// TIA Portal project "winda" (V17)

(* hardware
DEVICE "S7-1500/ET200MP station_1"  S7-1500 station
   slot 0: "Rail_0"  Rack  6ES7 590-1***0-0AA0
   slot 1: "PLC_1"  CPU 1513-1 PN  6ES7 513-1AL02-0AB0  V2.9
      slot 3: "CPU display_1"  6ES7591-1AA00-0AA0
      slot 32768: "PROFINET interface_1"  X1
         slot 32769: "Port_1"  X1 P1
         slot 32770: "Port_2"  X1 P2
      slot 34817: "Virtual CP interface port_1"  Virtual CP interface port  Virtual CP interface port
*)

// ===== PLC "PLC_1"  CPU 1513-1 PN =====

VAR_GLOBAL   // PLC tag table "Default tag table"
   "wybrane" AT %MW50 : Int;
   "aktualne" AT %MW52 : Int;
   "jazda_dol" AT %Q0.0 : Bool;
   "jazda_gora" AT %Q0.1 : Bool;
   "Tag_5" AT %M50.0 : Bool;
   "Tag_6" AT %I0.0 : Bool;
   "Tag_7" AT %I0.1 : Bool;
   "Tag_8" AT %I0.2 : Bool;
   "Tag_9" AT %I0.3 : Bool;
   "Tag_10" AT %MW51 : Int;
   "T1Q" AT %M54.0 : Bool;
   "Tag_1" AT %M54.1 : Bool;
END_VAR

DATA_BLOCK "winda_LAD_DB"   // DB3
{ S7_Optimized_Access := 'TRUE' }
VERSION : 0.1
// stored: InstanceOfName winda_LAD
"winda_LAD"
BEGIN
END_DATA_BLOCK

DATA_BLOCK "winda_graph_DB1"   // DB4
{ S7_Optimized_Access := 'TRUE' }
VERSION : 0.1
// stored: InstanceOfName winda_graph
"winda_graph"
BEGIN
END_DATA_BLOCK

// folder: System blocks/Program resources

DATA_BLOCK "IEC_Timer_0_DB_1"   // DB1
{ S7_Optimized_Access := 'TRUE' }
AUTHOR : Simatic
FAMILY : IEC
NAME : IEC_TMR
VERSION : 1.0
// stored: InstanceOfName IEC_TIMER
"IEC_TIMER"
BEGIN
END_DATA_BLOCK

DATA_BLOCK "IEC_Timer_0_DB"   // DB2
{ S7_Optimized_Access := 'TRUE' }
AUTHOR : Simatic
FAMILY : IEC
NAME : IEC_TMR
VERSION : 1.0
// stored: InstanceOfName IEC_TIMER
"IEC_TIMER"
BEGIN
END_DATA_BLOCK

DATA_BLOCK "IEC_Timer_0_DB_2"   // DB5
{ S7_Optimized_Access := 'TRUE' }
AUTHOR : Simatic
FAMILY : IEC
NAME : IEC_TMR
VERSION : 1.0
// stored: InstanceOfName IEC_TIMER
"IEC_TIMER"
BEGIN
END_DATA_BLOCK

// folder: (top level)

FUNCTION_BLOCK "winda_graph"   // FB1, GRAPH_PLUS
{ S7_Optimized_Access := 'TRUE' }
VERSION : 0.1
   VAR_INPUT
      OFF_SQ : Bool := false;   // Turn sequence off
      INIT_SQ : Bool := false;   // Set sequence to initial state
      ACK_EF : Bool := false;   // Acknowledge all errors and faults
      S_PREV : Bool := false;   // Output previous step in parameter S_NO
      S_NEXT : Bool := false;   // Indicate next step in parameter S_NO
      SW_AUTO : Bool := false;   // Automatic mode
      SW_TAP : Bool := false;   // Semiautomatic/switch with transition
      SW_TOP : Bool := false;   // Semiautomatic/ignore transition
      SW_MAN : Bool := false;   // Manual mode
      S_SEL : Int := 0;   // Select step to be output to S_NO
      S_ON : Bool := false;   // Activate step indicated in S_NO
      S_OFF : Bool := false;   // Deactivate step indicated S_NO
      T_PUSH : Bool := false;   // Enable transition to switch in semi automatic mode
      aktualne_pietro : Int;
      wybrane_pietro : Int;
   END_VAR
   VAR_OUTPUT
      S_NO : Int := 0;   // Step number
      S_MORE : Bool := false;   // More steps are available and can be shown in S_NO
      S_ACTIVE : Bool := false;   // Step indicated in S_NO is active
      ERR_FLT : Bool := false;   // Interlock or supervision group error
      AUTO_ON : Bool := false;   // Automatic mode is active
      TAP_ON : Bool := false;   // Semiautomatic mode/step with transition enabled
      TOP_ON : Bool := false;   // Semiautomatic mode/ignore transition enabled
      MAN_ON : Bool := false;   // Manual mode is active
   END_VAR
   VAR_IN_OUT
      jedz_dol : Bool;
      jedz_gora : Bool;
   END_VAR
   VAR
      HMI_INFO : Array[0..8] of UInt;
      IF_PAR : G7_IfParPlus_V6;
      RT_DATA : G7_RTDataPlus_V6;   // Internal data area
      Trans1 : G7_TransitionPlus_V6;   // Transition structure
      Trans2 : G7_TransitionPlus_V6;   // Transition structure
      Trans3 : G7_TransitionPlus_V6;   // Transition structure
      Trans4 : G7_TransitionPlus_V6;   // Transition structure
      Trans6 : G7_TransitionPlus_V6;   // Transition structure
      Trans8 : G7_TransitionPlus_V6;   // Transition structure
      START : G7_StepPlus_V6;   // Step structure
      JAZDA_GORA : G7_StepPlus_V6;   // Step structure
      STOP_WINDY : G7_StepPlus_V6;   // Step structure
      JAZDA_DOL : G7_StepPlus_V6;   // Step structure
      STOP_WINDY2 : G7_StepPlus_V6;   // Step structure
      SINI : Array[0..1] of USInt;
      LSTT : Array[0..5] of USInt;
      ATAJ : Array[0..5] of USInt;
      ATAB : Array[0..5] of USInt;
      PSTT : Array[0..5] of USInt;
      NSTT : Array[0..5] of USInt;
      ASSJ : Array[0..4] of USInt;
      ASSB : Array[0..4] of USInt;
      PTTS : Array[0..4] of USInt;
      NTTS : Array[0..4] of USInt;
      SW_SQTS : Array[0..4] of USInt;
      SWITCH : Array[0..1] of USInt;
      TVX : Array[0..3] of USInt;
      TTX : Array[0..3] of USInt;
      TSX : Array[0..1] of USInt;
      S00X : Array[0..1] of USInt;
      SOFFX : Array[0..1] of USInt;
      SONX : Array[0..1] of USInt;
      SAX : Array[0..1] of USInt;
      SERRX : Array[0..5] of USInt;
      SMX : Array[0..5] of USInt;
      S0X : Array[0..5] of USInt;
      S1X : Array[0..5] of USInt;
      IL_ALARM_INST : Diag_Alarm;
      SUP_ALARM_INST : Diag_Alarm;
      STEP_TIME_ALARM_INST : Diag_Alarm;
      IEC_TIMER_INST : IEC_TIMER;
      TRANSACTION_FLAG : Bool := false;
   END_VAR
   // SINI[0] := 2;
   // LSTT[0] := 255;
   // LSTT[1] := 255;
   // LSTT[2] := 255;
   // LSTT[4] := 255;
   // ATAJ[1] := 1;
   // ATAJ[2] := 2;
   // ATAJ[3] := 3;
   // ATAJ[4] := 4;
   // ATAJ[5] := 5;
   // ATAB[0] := 1;
   // ATAB[2] := 2;
   // ATAB[3] := 3;
   // ATAB[4] := 4;
   // ATAB[5] := 5;
   // PSTT[2] := 1;
   // PSTT[3] := 2;
   // PSTT[4] := 3;
   // PSTT[5] := 4;
   // NSTT[0] := 3;
   // NSTT[1] := 1;
   // NSTT[2] := 2;
   // NSTT[4] := 4;
   // ASSJ[1] := 1;
   // ASSJ[2] := 2;
   // ASSJ[3] := 3;
   // ASSJ[4] := 4;
   // ASSB[1] := 1;
   // ASSB[2] := 2;
   // ASSB[3] := 3;
   // ASSB[4] := 4;
   // PTTS[0] := 255;
   // PTTS[1] := 1;
   // PTTS[2] := 2;
   // PTTS[4] := 4;
   // NTTS[1] := 2;
   // NTTS[2] := 3;
   // NTTS[3] := 4;
   // NTTS[4] := 5;
   // SW_SQTS[1] := 1;
   // SW_SQTS[2] := 1;
   // SW_SQTS[3] := 2;
   // SW_SQTS[4] := 2;
   // TVX[0] := 16#1;
   // TTX[0] := 16#1;
   // TSX[0] := 16#1;
   // S00X[0] := 16#1;
   // SOFFX[0] := 16#1;
   // SONX[0] := 16#1;
   // SAX[0] := 16#1;
   // SERRX[0] := 16#1;
   // SMX[0] := 16#1;
   // S0X[0] := 16#1;
   // S1X[0] := 16#1;
BEGIN
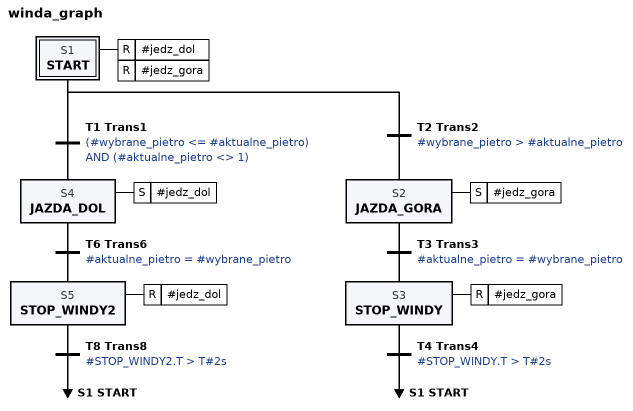
   // sequencer 1
   INITIAL_STEP START:   // S1, max time T#10S, warning time T#7S
              R    #jedz_dol
              R    #jedz_gora
   END_STEP
   TRANSITION Trans1 FROM START TO JAZDA_DOL   // T1
      := (#wybrane_pietro <= #aktualne_pietro) AND (#aktualne_pietro <> 1);
   END_TRANSITION
   TRANSITION Trans2 FROM START TO JAZDA_GORA   // T2
      := #wybrane_pietro > #aktualne_pietro;
   END_TRANSITION
   STEP JAZDA_GORA:   // S2, max time T#10S, warning time T#7S
              S    #jedz_gora
   END_STEP
   TRANSITION Trans3 FROM JAZDA_GORA TO STOP_WINDY   // T3
      := #aktualne_pietro = #wybrane_pietro;
   END_TRANSITION
   STEP STOP_WINDY:   // S3, max time T#10S, warning time T#7S
              R    #jedz_gora
   END_STEP
   TRANSITION Trans4 FROM STOP_WINDY TO START   // T4, jump
      := #STOP_WINDY.T > T#2s;
   END_TRANSITION
   STEP JAZDA_DOL:   // S4, max time T#10S, warning time T#7S
              S    #jedz_dol
   END_STEP
   TRANSITION Trans6 FROM JAZDA_DOL TO STOP_WINDY2   // T6
      := #aktualne_pietro = #wybrane_pietro;
   END_TRANSITION
   STEP STOP_WINDY2:   // S5, max time T#10S, warning time T#7S
              R    #jedz_dol
   END_STEP
   TRANSITION Trans8 FROM STOP_WINDY2 TO START   // T8, jump
      := #STOP_WINDY2.T > T#2s;
   END_TRANSITION
END_FUNCTION_BLOCK

FUNCTION_BLOCK "winda_LAD"   // FB2, LAD
{ S7_Optimized_Access := 'TRUE' }
VERSION : 0.1
   VAR_INPUT
      "1" : Bool;
      "2" : Bool;
      "3" : Bool;
      "4" : Bool;
   END_VAR
   VAR_IN_OUT
      aktualne_pietro : Int := 1;
      wybrane_pietro : Int := 1;
      jedz_dol : Bool;
      jedz_gora : Bool;
   END_VAR
   VAR
      START : Bool;
      JAZDA_DOL : Bool;
      JAZDA_GORA : Bool;
      "STOP WINDY" : Bool;
      kolejka : Array[0..3] of Bool;
      "1_static" : Bool;
      "2_static" : Bool;
      "3_static" : Bool;
      "4_static" : Bool;
   END_VAR
   VAR_TEMP
      v : Int;
   END_VAR
   VAR_TEMP   // added for the SCL form of the ladder/FBD networks
      _w1 : Bool;
      _w2 : Bool;
      _w3 : Bool;
      _w4 : Bool;
   END_VAR
BEGIN

REGION Network 1
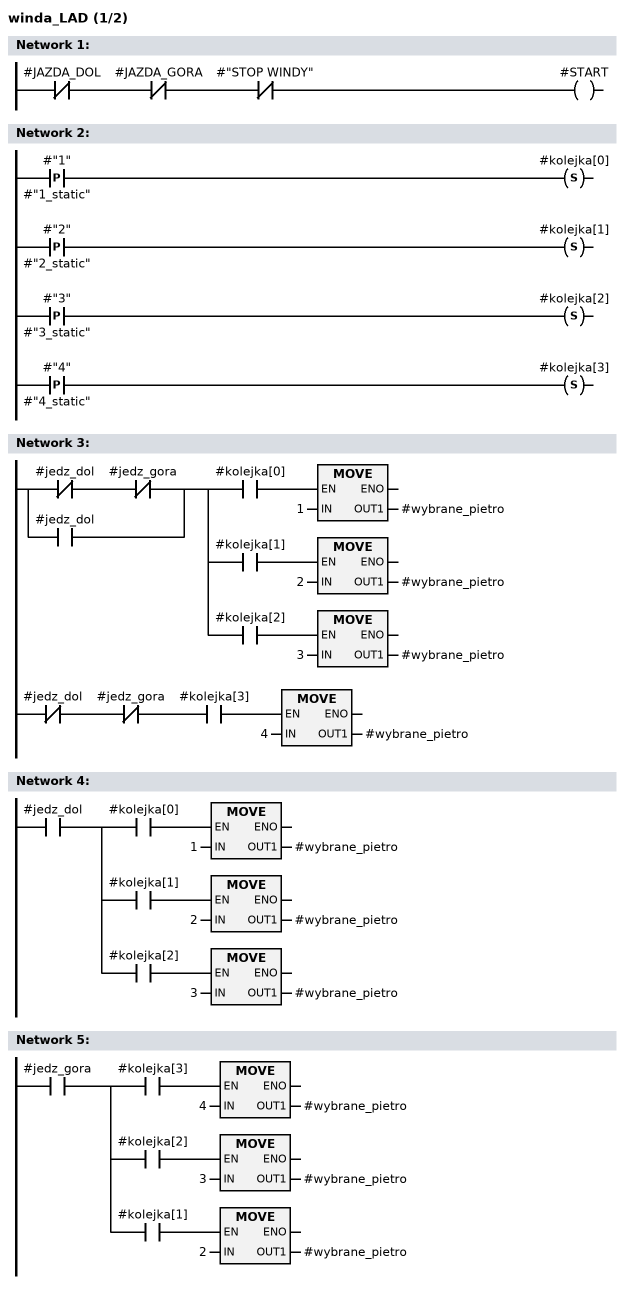
   RUNG wire#powerrail
      I_Contact( #JAZDA_DOL )
      I_Contact( #JAZDA_GORA )
      I_Contact( #"STOP WINDY" )
      Coil( #START )
   END_RUNG
   // the same network as SCL:
   #START := NOT #JAZDA_DOL AND NOT #JAZDA_GORA AND NOT #"STOP WINDY";
END_REGION

REGION Network 2
   RUNG wire#powerrail
      P_Contact(operand := #"1", bit := #"1_static")
      S_Coil( #kolejka[0] )
   END_RUNG
   RUNG wire#powerrail
      P_Contact(operand := #"2", bit := #"2_static")
      S_Coil( #kolejka[1] )
   END_RUNG
   RUNG wire#powerrail
      P_Contact(operand := #"3", bit := #"3_static")
      S_Coil( #kolejka[2] )
   END_RUNG
   RUNG wire#powerrail
      P_Contact(operand := #"4", bit := #"4_static")
      S_Coil( #kolejka[3] )
   END_RUNG
   // the same network as SCL:
   #_w1 := #"1" AND NOT #"1_static";   // rising edge of #"1"
   #"1_static" := #"1";
   IF #_w1 THEN #kolejka[0] := TRUE; END_IF;
   #_w2 := #"2" AND NOT #"2_static";   // rising edge of #"2"
   #"2_static" := #"2";
   IF #_w2 THEN #kolejka[1] := TRUE; END_IF;
   #_w3 := #"3" AND NOT #"3_static";   // rising edge of #"3"
   #"3_static" := #"3";
   IF #_w3 THEN #kolejka[2] := TRUE; END_IF;
   #_w4 := #"4" AND NOT #"4_static";   // rising edge of #"4"
   #"4_static" := #"4";
   IF #_w4 THEN #kolejka[3] := TRUE; END_IF;
END_REGION

REGION Network 3
   RUNG wire#powerrail
      I_Contact( #jedz_dol )
      I_Contact( #jedz_gora )
      wire#w1
      Contact( #kolejka[0] )
      Move(in := 1, out1 => #wybrane_pietro)
   END_RUNG
   RUNG wire#powerrail
      Contact( #jedz_dol )
   END_RUNG wire#w1
   RUNG wire#w1
      Contact( #kolejka[1] )
      Move(in := 2, out1 => #wybrane_pietro)
   END_RUNG
   RUNG wire#w1
      Contact( #kolejka[2] )
      Move(in := 3, out1 => #wybrane_pietro)
   END_RUNG
   RUNG wire#powerrail
      I_Contact( #jedz_dol )
      I_Contact( #jedz_gora )
      Contact( #kolejka[3] )
      Move(in := 4, out1 => #wybrane_pietro)
   END_RUNG
   // the same network as SCL:
   #_w1 := (NOT #jedz_dol AND NOT #jedz_gora) OR #jedz_dol;
   IF #_w1 AND #kolejka[0] THEN #wybrane_pietro := 1; END_IF;
   IF #_w1 AND #kolejka[1] THEN #wybrane_pietro := 2; END_IF;
   IF #_w1 AND #kolejka[2] THEN #wybrane_pietro := 3; END_IF;
   IF NOT #jedz_dol AND NOT #jedz_gora AND #kolejka[3] THEN #wybrane_pietro := 4; END_IF;
END_REGION

REGION Network 4
   RUNG wire#powerrail
      Contact( #jedz_dol )
      wire#w1
      Contact( #kolejka[0] )
      Move(in := 1, out1 => #wybrane_pietro)
   END_RUNG
   RUNG wire#w1
      Contact( #kolejka[1] )
      Move(in := 2, out1 => #wybrane_pietro)
   END_RUNG
   RUNG wire#w1
      Contact( #kolejka[2] )
      Move(in := 3, out1 => #wybrane_pietro)
   END_RUNG
   // the same network as SCL:
   IF #jedz_dol AND #kolejka[0] THEN #wybrane_pietro := 1; END_IF;
   IF #jedz_dol AND #kolejka[1] THEN #wybrane_pietro := 2; END_IF;
   IF #jedz_dol AND #kolejka[2] THEN #wybrane_pietro := 3; END_IF;
END_REGION

REGION Network 5
   RUNG wire#powerrail
      Contact( #jedz_gora )
      wire#w1
      Contact( #kolejka[3] )
      Move(in := 4, out1 => #wybrane_pietro)
   END_RUNG
   RUNG wire#w1
      Contact( #kolejka[2] )
      Move(in := 3, out1 => #wybrane_pietro)
   END_RUNG
   RUNG wire#w1
      Contact( #kolejka[1] )
      Move(in := 2, out1 => #wybrane_pietro)
   END_RUNG
   // the same network as SCL:
   IF #jedz_gora AND #kolejka[3] THEN #wybrane_pietro := 4; END_IF;
   IF #jedz_gora AND #kolejka[2] THEN #wybrane_pietro := 3; END_IF;
   IF #jedz_gora AND #kolejka[1] THEN #wybrane_pietro := 2; END_IF;
END_REGION

REGION Network 6
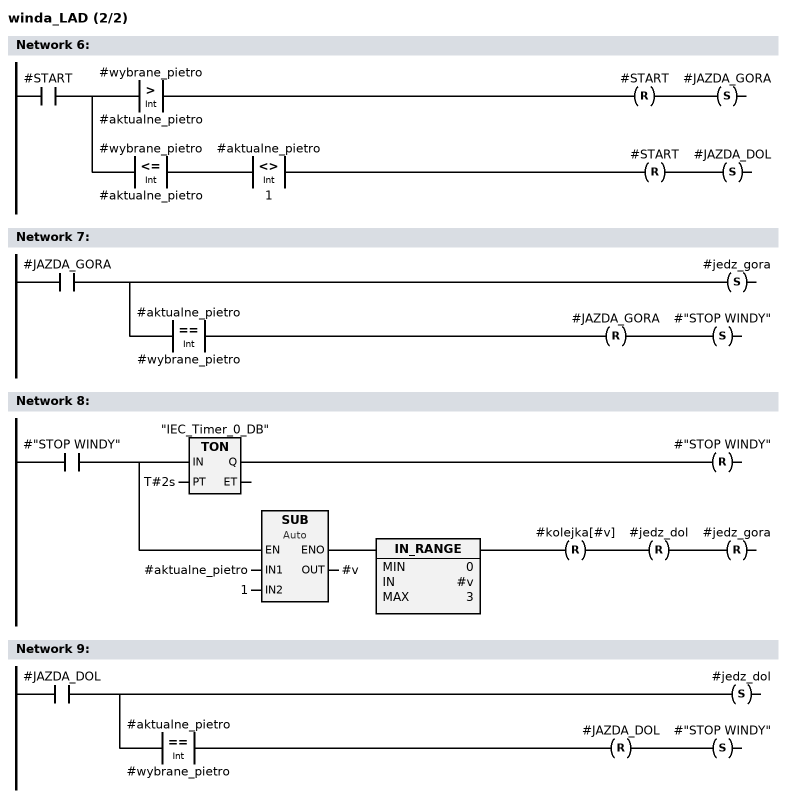
   RUNG wire#powerrail
      Contact( #START )
      wire#w1
      { S7_Templates := "SrcType := Int" } GT_Contact(in1 := #wybrane_pietro, in2 := #aktualne_pietro)
      R_Coil( #START )
      S_Coil( #JAZDA_GORA )
   END_RUNG
   RUNG wire#w1
      { S7_Templates := "SrcType := Int" } LE_Contact(in1 := #wybrane_pietro, in2 := #aktualne_pietro)
      { S7_Templates := "SrcType := Int" } NE_Contact(in1 := #aktualne_pietro, in2 := 1)
      R_Coil( #START )
      S_Coil( #JAZDA_DOL )
   END_RUNG
   // the same network as SCL:
   #_w1 := #START AND (#wybrane_pietro > #aktualne_pietro);
   #_w2 := #START;
   IF #_w1 THEN
       #START := FALSE;
       #JAZDA_GORA := TRUE;
   END_IF;
   IF #_w2 AND (#wybrane_pietro <= #aktualne_pietro) AND (#aktualne_pietro <> 1) THEN
       #START := FALSE;
       #JAZDA_DOL := TRUE;
   END_IF;
END_REGION

REGION Network 7
   RUNG wire#powerrail
      Contact( #JAZDA_GORA )
      wire#w1
      S_Coil( #jedz_gora )
   END_RUNG
   RUNG wire#w1
      { S7_Templates := "SrcType := Int" } EQ_Contact(in1 := #aktualne_pietro, in2 := #wybrane_pietro)
      R_Coil( #JAZDA_GORA )
      S_Coil( #"STOP WINDY" )
   END_RUNG
   // the same network as SCL:
   IF #JAZDA_GORA THEN #jedz_gora := TRUE; END_IF;
   #_w1 := #JAZDA_GORA AND (#aktualne_pietro = #wybrane_pietro);
   IF #_w1 THEN
       #JAZDA_GORA := FALSE;
       #"STOP WINDY" := TRUE;
   END_IF;
END_REGION

REGION Network 8
   "IEC_Timer_0_DB".TON(IN := #"STOP WINDY", PT := T#2s);
   #_w1 := #"STOP WINDY";
   IF "IEC_Timer_0_DB".Q THEN #"STOP WINDY" := FALSE; END_IF;
   IF #_w1 THEN #v := #aktualne_pietro - 1; END_IF;
   #_w2 := #_w1 AND (0 <= #v) AND (#v <= 3);
   IF #_w2 THEN
       #kolejka[#v] := FALSE;
       #jedz_dol := FALSE;
       #jedz_gora := FALSE;
   END_IF;
END_REGION

REGION Network 9
   RUNG wire#powerrail
      Contact( #JAZDA_DOL )
      wire#w1
      S_Coil( #jedz_dol )
   END_RUNG
   RUNG wire#w1
      { S7_Templates := "SrcType := Int" } EQ_Contact(in1 := #aktualne_pietro, in2 := #wybrane_pietro)
      R_Coil( #JAZDA_DOL )
      S_Coil( #"STOP WINDY" )
   END_RUNG
   // the same network as SCL:
   IF #JAZDA_DOL THEN #jedz_dol := TRUE; END_IF;
   #_w1 := #JAZDA_DOL AND (#aktualne_pietro = #wybrane_pietro);
   IF #_w1 THEN
       #JAZDA_DOL := FALSE;
       #"STOP WINDY" := TRUE;
   END_IF;
END_REGION
END_FUNCTION_BLOCK

ORGANIZATION_BLOCK "Main"   // OB1, LAD, ProgramCycle
TITLE = "Main Program Sweep (Cycle)"
{ S7_Optimized_Access := 'TRUE' }
VERSION : 0.1
   VAR_INPUT
      Initial_Call : Bool;   // Initial call of this OB
      Remanence : Bool;   // =True, if remanent data are available
   END_VAR
BEGIN

REGION Network 1
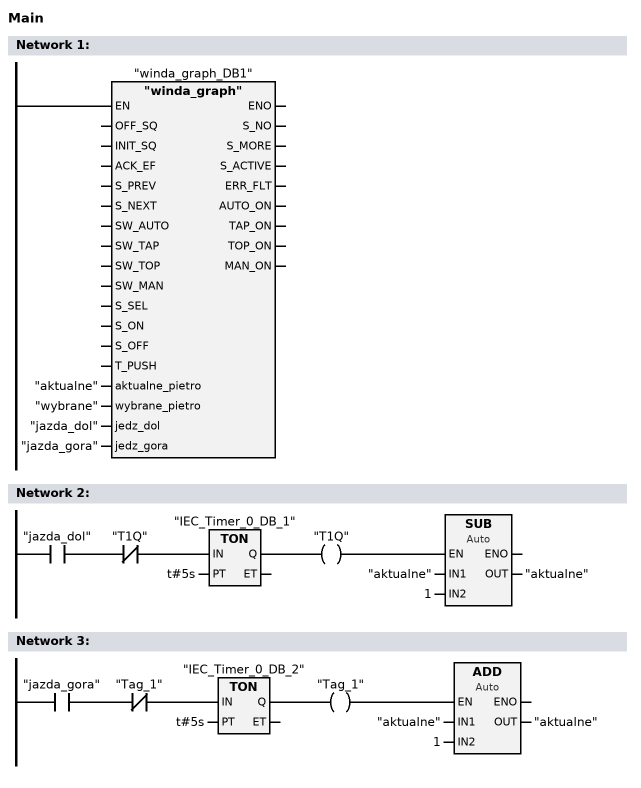
   RUNG wire#powerrail
      "winda_graph_DB1"(OFF_SQ :=, INIT_SQ :=, ACK_EF :=, S_PREV :=, S_NEXT :=, SW_AUTO :=, SW_TAP :=, SW_TOP :=, SW_MAN :=, S_SEL :=, S_ON :=, S_OFF :=, T_PUSH :=, aktualne_pietro := "aktualne", wybrane_pietro := "wybrane", jedz_dol := "jazda_dol", jedz_gora := "jazda_gora", S_NO =>, S_MORE =>, S_ACTIVE =>, ERR_FLT =>, AUTO_ON =>, TAP_ON =>, TOP_ON =>, MAN_ON =>)
   END_RUNG
   // the same network as SCL:
   "winda_graph_DB1"(aktualne_pietro := "aktualne",   // "winda_graph"
                     wybrane_pietro := "wybrane",
                     jedz_dol := "jazda_dol",
                     jedz_gora := "jazda_gora");
END_REGION

REGION Network 2
   "IEC_Timer_0_DB_1".TON(IN := "jazda_dol" AND NOT "T1Q", PT := t#5s);
   "T1Q" := "IEC_Timer_0_DB_1".Q;
   IF "IEC_Timer_0_DB_1".Q THEN "aktualne" := "aktualne" - 1; END_IF;
END_REGION

REGION Network 3
   "IEC_Timer_0_DB_2".TON(IN := "jazda_gora" AND NOT "Tag_1", PT := t#5s);
   "Tag_1" := "IEC_Timer_0_DB_2".Q;
   IF "IEC_Timer_0_DB_2".Q THEN "aktualne" := "aktualne" + 1; END_IF;
END_REGION
END_ORGANIZATION_BLOCK

ORGANIZATION_BLOCK "Startup"   // OB100, LAD, Startup
TITLE = "Complete Restart"
{ S7_Optimized_Access := 'TRUE' }
VERSION : 0.1
   VAR_INPUT
      LostRetentive : Bool;   // True if retentive data are lost
      LostRTC : Bool;   // True if date and time are lost
   END_VAR
BEGIN

REGION Network 1
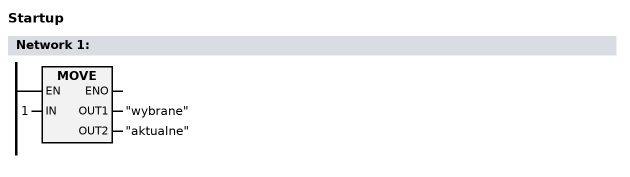
   RUNG wire#powerrail
      Move(in := 1, out1 => "wybrane", out2 => "aktualne")
   END_RUNG
   // the same network as SCL:
   "wybrane" := 1;
   "aktualne" := 1;
END_REGION
END_ORGANIZATION_BLOCK